// ---- VISUs/SETTING/SettingArm_Page.TcVIS
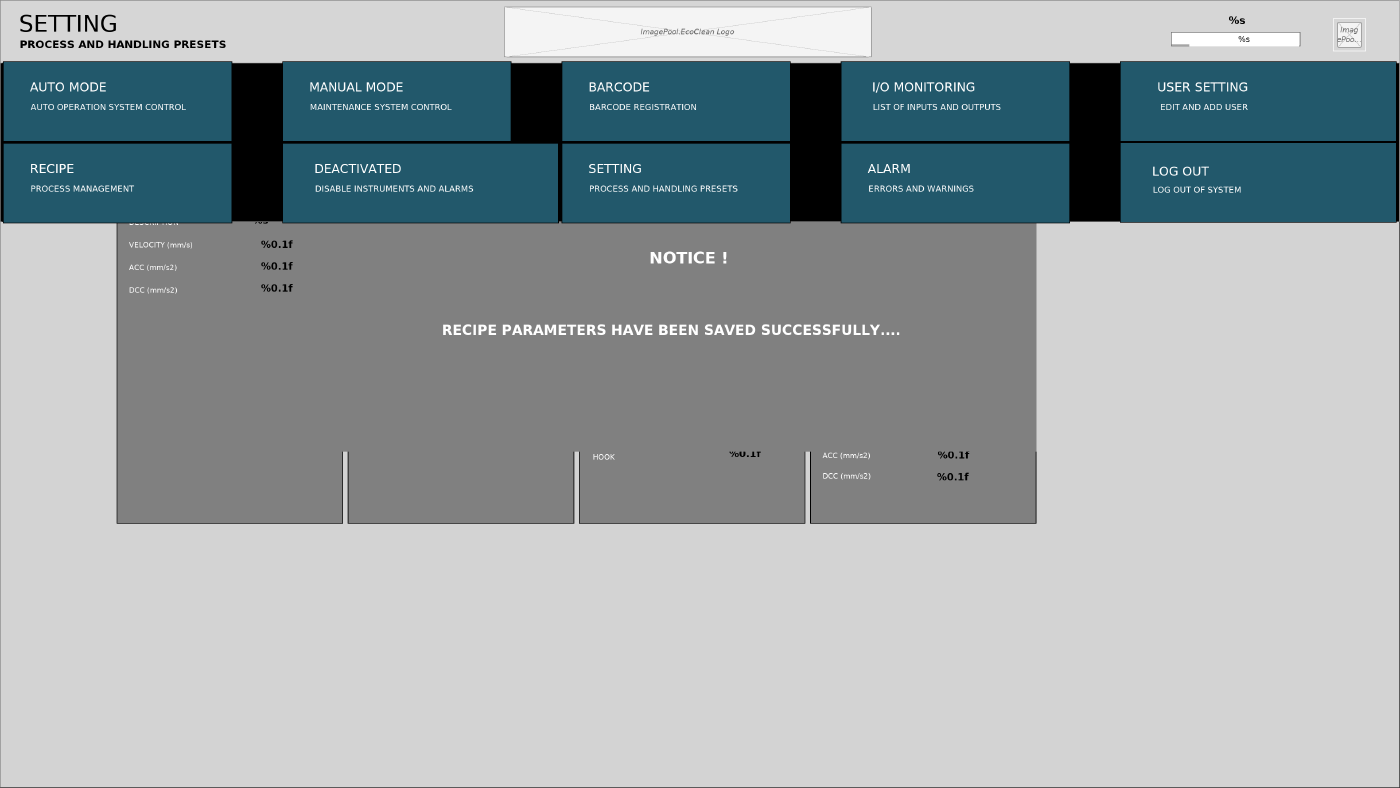
VISUALIZATION SettingArm_Page  // 1920x1081
    Rectangle (0,101 1920x980)
    Rectangle (0,63 1920x26)
        p3528305787: HMI_Ctrl.ANIMATION3
    Rectangle (0,0 1919x85)
    Label (23,6 267x53), "SETTING"
    Label (24,49 320x24), "PROCESS AND HANDLING PRESETS"
    Group (1828,25 45x45)
        OnMouseClick: toggle HMI_Ctrl.MenuButton
        RoundedRectangle (0,0 45x45), colour toggle: HMI_Ctrl.MenuButton
        Image (6,5 33x35), image: ImagePool.Menu Button
    Ellipse (867,123 25x25)
    Ellipse (948,123 25x25)
    Ellipse (904,130 10x10)
    Ellipse (926,130 10x10)
    Ellipse (985,130 10x10)
    Ellipse (1007,130 10x10)
    Ellipse (1029,123 25x25)
    Label (847,153 64x24), "BASIC"
    Label (928,153 64x24), "PROCESS"
    Label (1009,153 64x24), "ARM"
    Image (790,113 45x45), image: ImagePool.Previous Button
        OnMouseClick: change screen: SettingProcess_Page
    RoundedRectangle (1441,125 314x48)
    ComboBoxInteger (1555,132 189x37), variable: iArmSettingStnNoBuffer, text list: 'TextList_Arm_Setting'
    Label (1461,141 79x24), "STATION"
    Rectangle (160,218 310x500)
    Rectangle (160,219 310x27)
    Label (178,222 143x24), "ARM SPEED PROFILE"
    Label (174,262 141x24), "SPEED PROFILE NO."
    Label (174,293 108x24), "DESCRIPTION"
    Label (174,324 116x24), "VELOCITY (mm/s)"
    Label (174,355 118x24), "ACC (mm/s2)"
    Label (174,386 82x24), "DCC (mm/s2)"
    Rectangle (477,218 310x500)
    Rectangle (477,219 310x27)
    Label (495,222 213x24), "ARM UP AND DOWN PATTERN"
    Rectangle (794,218 310x500)
    Rectangle (794,219 310x27)
    Label (812,222 228x24), "ARM VERTICAL POSITION (MM)"
    Rectangle (1111,218 310x500)
    Rectangle (1111,219 310x27)
    Label (1129,222 200x24), "ARM VERTICAL SETTING"
    Label (1125,262 109x24), "1st VELO (mm/s)"
    Label (1125,293 108x24), "ACC (mm/s2)"
    Label (491,262 147x24), "SPEED PATTERN NO"
    Label (491,293 108x24), "DESCRIPTION"
    Label (491,324 196x24), "1ST STAGE SPEED PROFILE"
    Label (491,355 186x24), "2ND STAGE SPEED PROFILE"
    Label (491,391 186x24), "3RD STAGE SPEED PROFILE"
    Label (491,427 186x24), "4TH STAGE SPEED PROFILE"
    Label (808,262 147x24), "TOP POSITION"
    Label (808,293 108x24), "1ST STAGE"
    Label (808,324 196x24), "2ND STAGE"
    Label (808,355 186x24), "3RD STAGE"
    Label (808,386 186x24), "4TH STAGE"
    Label (808,427 186x24), "BOTTOM POSITION"
    Rectangle (1111,539 310x27)
    Label (1129,541 200x24), "ARM HORIZONTAL SETTING"
    Rectangle (310,267 140x17), "%i", text variable: DSA31ArmSpeedProfileStore.iArmSpdProfileNo, input disabled if: bMainOnOff
        OnMouseDown: write the text variable via VisuDialogs.Numpad, min 1, max 20
    Rectangle (263,294 189x17), "%s", text variable: DSA31ArmSpeedProfileStore.DsArmSpeedProfile.sDescription, input disabled if: bMainOnOff
        OnMouseDown: write the text variable via VisuDialogs.Keypad
    Rectangle (310,327 140x17), "%0.1f", text variable: DSA31ArmSpeedProfileStore.DsArmSpeedProfile.lrSpeedVelo, input disabled if: bMainOnOff
        OnMouseDown: write the text variable via VisuDialogs.Numpad, min 2, max 400
    Rectangle (310,357 140x17), "%0.1f", text variable: DSA31ArmSpeedProfileStore.DsArmSpeedProfile.lrAcc, input disabled if: bMainOnOff
        OnMouseDown: write the text variable via VisuDialogs.Numpad, min 100, max 1500
    Rectangle (310,387 140x17), "%0.1f", text variable: DSA31ArmSpeedProfileStore.DsArmSpeedProfile.lrDcc, input disabled if: bMainOnOff
        OnMouseDown: write the text variable via VisuDialogs.Numpad, min 100, max 1500
    Rectangle (653,264 131x17), "%i", text variable: DSA21UpDownPatternStore.iUpDownPatternNo, input disabled if: bMainOnOff
        OnMouseDown: write the text variable via VisuDialogs.Numpad, min 1, max 20
    Rectangle (654,325 129x17), "%i", text variable: DSA21UpDownPatternStore.DsInUpDownPatternMemory.iZone1SpdProfileNo, input disabled if: bMainOnOff
        OnMouseDown: write the text variable via VisuDialogs.Numpad, min 1, max 20
    Rectangle (654,360 129x17), "%i", text variable: DSA21UpDownPatternStore.DsInUpDownPatternMemory.iZone2SpdProfileNo, input disabled if: bMainOnOff
        OnMouseDown: write the text variable via VisuDialogs.Numpad, min 1, max 20
    Rectangle (654,400 129x17), "%i", text variable: DSA21UpDownPatternStore.DsInUpDownPatternMemory.iZone3SpdProfileNo, input disabled if: bMainOnOff
        OnMouseDown: write the text variable via VisuDialogs.Numpad, min 1, max 20
    Rectangle (654,432 129x17), "%i", text variable: DSA21UpDownPatternStore.DsInUpDownPatternMemory.iZone4SpdProfileNo, input disabled if: bMainOnOff
        OnMouseDown: write the text variable via VisuDialogs.Numpad, min 1, max 20
    Rectangle (583,294 189x17), "%s", text variable: DSA21UpDownPatternStore.DsInUpDownPatternMemory.sDescription, input disabled if: bMainOnOff
        OnMouseDown: write the text variable via VisuDialogs.Keypad
    Rectangle (951,264 140x17), "%0.1f", text variable: Arm1TopPos[iArmSettingStnNo], input disabled if: bMainOnOff
        OnMouseDown: write the text variable via VisuDialogs.Numpad
    Rectangle (951,294 140x17), "%0.1f", text variable: Arm1Pos1stStage[iArmSettingStnNo], input disabled if: bMainOnOff
        OnMouseDown: write the text variable via VisuDialogs.Numpad
    Rectangle (951,324 140x17), "%0.1f", text variable: Arm1Pos2ndStage[iArmSettingStnNo], input disabled if: bMainOnOff
        OnMouseDown: write the text variable via VisuDialogs.Numpad
    Rectangle (951,354 140x17), "%0.1f", text variable: Arm1Pos3rdStage[iArmSettingStnNo], input disabled if: bMainOnOff
        OnMouseDown: write the text variable via VisuDialogs.Numpad
    Rectangle (951,389 140x17), "%0.1f", text variable: Arm1Pos4thStage[iArmSettingStnNo], input disabled if: bMainOnOff
        OnMouseDown: write the text variable via VisuDialogs.Numpad
    Rectangle (951,424 140x17), "%0.1f", text variable: Arm1BottomPos[iArmSettingStnNo], input disabled if: bMainOnOff
        OnMouseDown: write the text variable via VisuDialogs.Numpad
    Rectangle (794,539 310x27)
    Label (811,541 228x24), "ARM HORIZONTAL POSITION (MM)"
    Label (810,584 109x24), "UNHOOK"
    Label (810,615 108x24), "HOOK"
    Rectangle (951,584 140x17), "%0.1f", text variable: Arm1UnHookPos[iArmSettingStnNo], input disabled if: bMainOnOff
        OnMouseDown: write the text variable via VisuDialogs.Numpad
    Rectangle (952,614 140x17), "%0.1f", text variable: Arm1HookPos[iArmSettingStnNo], input disabled if: bMainOnOff
        OnMouseDown: write the text variable via VisuDialogs.Numpad
    Label (1125,321 108x24), "DCC (mm/s2)"
    Rectangle (1237,266 140x17), "%0.1f", text variable: ARlrVertPos_In_HighSpeed[1], input disabled if: bMainOnOff
        OnMouseDown: write the text variable via VisuDialogs.Numpad, min 2, max 400
    Rectangle (1238,296 140x17), "%0.1f", text variable: ARlrVertPos_In_Acc[1], input disabled if: bMainOnOff
        OnMouseDown: write the text variable via VisuDialogs.Numpad, min 200, max 1500
    Rectangle (1237,326 140x17), "%0.1f", text variable: ARlrVertPos_In_Dcc[1], input disabled if: bMainOnOff
        OnMouseDown: write the text variable via VisuDialogs.Numpad, min 200, max 1500
    Label (1125,582 109x24), "1st VELO (mm/s)"
    Label (1125,613 108x24), "ACC (mm/s2)"
    Label (1125,641 108x24), "DCC (mm/s2)"
    Rectangle (1237,586 140x17), "%0.1f", text variable: ARlrHorzPos_In_HighSpeed[1], input disabled if: bMainOnOff
        OnMouseDown: write the text variable via VisuDialogs.Numpad, min 50, max 600
    Rectangle (1238,616 140x17), "%0.1f", text variable: ARlrHorzPos_In_Acc[1], input disabled if: bMainOnOff
        OnMouseDown: write the text variable via VisuDialogs.Numpad, min 200, max 1500
    Rectangle (1237,646 140x17), "%0.1f", text variable: ARlrHorzPos_In_Dcc[1], input disabled if: bMainOnOff
        OnMouseDown: write the text variable via VisuDialogs.Numpad, min 200, max 1500
    Image (691,9 504x69), image: ImagePool.EcoClean Logo
    Label (808,465 186x24), "MID POSITION", invisible if: iArmSettingStnNo<>9
    Rectangle (951,469 140x17), "%0.1f", text variable: Arm1MidPos[iArmSettingStnNo], invisible if: iArmSettingStnNo<>9, input disabled if: bMainOnOff
        OnMouseDown: write the text variable via VisuDialogs.Numpad
    Group (1606,17 179x46)
        Button (0,27 177x19), image: VisuSymbols.Symbols.AddUser
        Rectangle (25,28 150x18), "%s", text variable: fbHmiTF1800_UserlevelManagement.dsHmiUserStatus_Active.sLoginName
        Rectangle (2,0 177x22), "%s", text variable: DSLocalSystemTimeML.sCurrentDT24Hr_General
    Group (1439,220 56x80), invisible if: bMainOnOff
        Label (5,52 51x28), "SAVE", invisible if: bMainOnOff
        RoundedRectangle (0,0 55x56), colour toggle: bRecipeSavePb
            tap bRecipeSavePb
        Image (11,5 34x45), image: ImagePool.Save Button
            OnMouseDown: execute { bRecipeSavePb:=1; }
            OnMouseUp: execute { bRecipeSavePb:=0; }
    Frame (457,253 964x366), invisible if: NOT stWritePersistentData.SaveHR
        shows Popup_Parameter_Saved()
    Frame (0,84 1918x221), invisible if: HMI_Ctrl.CloseMenuButton
        shows Popup_MenuPage()
END_VISUALIZATION

// ---- VISUs/SETTING/SettingProcess_Page.TcVIS
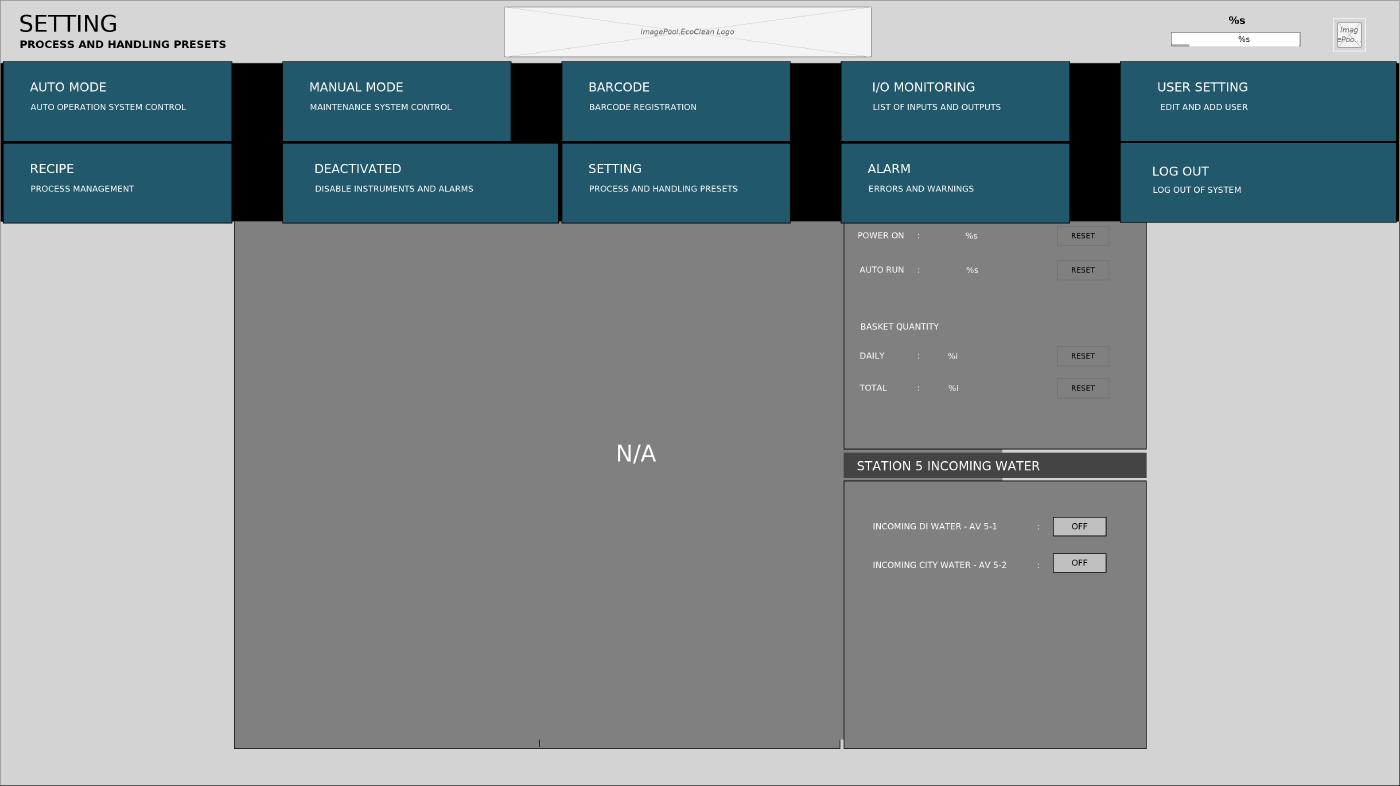
VISUALIZATION SettingProcess_Page  // 1920x1078
    Rectangle (0,101 1920x977)
    Rectangle (321,247 831x780)
    Rectangle (0,63 1920x26)
        p3528305787: HMI_Ctrl.ANIMATION3
    Rectangle (0,0 1919x85)
    Label (23,6 267x53), "SETTING"
    Label (24,49 320x24), "PROCESS AND HANDLING PRESETS"
    Group (1828,25 45x45)
        OnMouseClick: toggle HMI_Ctrl.MenuButton
        RoundedRectangle (0,0 45x45), colour toggle: HMI_Ctrl.MenuButton
        Image (6,5 33x35), image: ImagePool.Menu Button
    Ellipse (867,123 25x25)
    Ellipse (948,123 25x25)
    Ellipse (904,130 10x10)
    Ellipse (926,130 10x10)
    Ellipse (985,130 10x10)
    Ellipse (1007,130 10x10)
    Ellipse (1029,123 25x25)
    Label (847,153 64x24), "BASIC"
    Label (928,153 64x24), "PROCESS"
    Label (1009,153 64x24), "ARM"
    Image (1086,113 45x45), image: ImagePool.Next Button
        OnMouseClick: change screen: SettingArm_Page
    Image (790,113 45x45), image: ImagePool.Previous Button
        OnMouseClick: change screen: Setting_Page
    Rectangle (320,210 833x34)
    Label (582,217 283x24), "TIME OPTIMIZE/TRACKER"
    RoundedRectangle (491,308 30x30), colour toggle: ARbProductRecipeTimeBlockAvailable[1]
    RoundedRectangle (491,378 30x30), colour toggle: ARbProductRecipeTimeBlockAvailable[2]
    RoundedRectangle (491,446 30x30), colour toggle: ARbProductRecipeTimeBlockAvailable[3]
    RoundedRectangle (491,523 30x30), colour toggle: ARbProductRecipeTimeBlockAvailable[4]
    RoundedRectangle (491,598 30x30), colour toggle: ARbProductRecipeTimeBlockAvailable[5]
    RoundedRectangle (491,678 30x30), colour toggle: ARbProductRecipeTimeBlockAvailable[6]
    RoundedRectangle (491,758 30x30), colour toggle: ARbProductRecipeTimeBlockAvailable[7]
    RoundedRectangle (491,829 30x30), colour toggle: ARbProductRecipeTimeBlockAvailable[8]
    RoundedRectangle (491,898 30x30), colour toggle: ARbProductRecipeTimeBlockAvailable[9]
    Label (484,260 103x25), "ENABLE"
    RoundedRectangle (491,968 30x30), colour toggle: ARbProductRecipeTimeBlockAvailable[10]
    Label (385,307 37x24), "1"
    Label (385,377 37x24), "2"
    Label (385,445 37x24), "3"
    Label (385,522 37x24), "4"
    Label (385,597 37x24), "5"
    Label (385,677 37x24), "6"
    Label (385,757 37x24), "7"
    Label (385,828 37x24), "8"
    Label (385,897 37x24), "9"
    Label (380,967 37x24), "10"
    Label (360,248 113x46), "RECIPE NO"
    RoundedRectangle (594,306 90x40), "RESET", input disabled if: bMainOnOff
        tap bTrackerReset[1]
    RoundedRectangle (594,376 90x40), "RESET", input disabled if: bMainOnOff
        tap bTrackerReset[2]
    RoundedRectangle (594,444 90x40), "RESET", input disabled if: bMainOnOff
        tap bTrackerReset[3]
    RoundedRectangle (594,521 90x40), "RESET", input disabled if: bMainOnOff
        tap bTrackerReset[4]
    RoundedRectangle (594,596 90x40), "RESET", input disabled if: bMainOnOff
        tap bTrackerReset[5]
    RoundedRectangle (594,676 90x40), "RESET", input disabled if: bMainOnOff
        tap bTrackerReset[6]
    RoundedRectangle (594,756 90x40), "RESET", input disabled if: bMainOnOff
        tap bTrackerReset[7]
    RoundedRectangle (594,827 90x40), "RESET", input disabled if: bMainOnOff
        tap bTrackerReset[8]
    RoundedRectangle (594,896 90x40), "RESET", input disabled if: bMainOnOff
        tap bTrackerReset[9]
    RoundedRectangle (594,966 90x40), "RESET", input disabled if: bMainOnOff
        tap bTrackerReset[10]
    RoundedRectangle (906,308 30x30), colour toggle: ARbProductRecipeTimeBlockAvailable[11]
    RoundedRectangle (906,378 30x30), colour toggle: ARbProductRecipeTimeBlockAvailable[12]
    RoundedRectangle (906,446 30x30), colour toggle: ARbProductRecipeTimeBlockAvailable[13]
    RoundedRectangle (906,523 30x30), colour toggle: ARbProductRecipeTimeBlockAvailable[14]
    RoundedRectangle (906,598 30x30), colour toggle: ARbProductRecipeTimeBlockAvailable[15]
    RoundedRectangle (906,678 30x30), colour toggle: ARbProductRecipeTimeBlockAvailable[16]
    RoundedRectangle (906,758 30x30), colour toggle: ARbProductRecipeTimeBlockAvailable[17]
    RoundedRectangle (906,829 30x30), colour toggle: ARbProductRecipeTimeBlockAvailable[18]
    RoundedRectangle (906,898 30x30), colour toggle: ARbProductRecipeTimeBlockAvailable[19]
    Label (894,258 103x25), "ENABLE"
    RoundedRectangle (906,968 30x30), colour toggle: ARbProductRecipeTimeBlockAvailable[20]
    Label (803,309 37x24), "11"
    Label (803,379 37x24), "12"
    Label (803,447 37x24), "13"
    Label (803,524 37x24), "14"
    Label (803,599 37x24), "15"
    Label (803,679 37x24), "16"
    Label (803,759 37x24), "17"
    Label (803,830 37x24), "18"
    Label (803,899 37x24), "19"
    Label (802,969 37x24), "20"
    RoundedRectangle (1007,306 90x40), "RESET", input disabled if: bMainOnOff
        tap bTrackerReset[11]
    RoundedRectangle (1007,376 90x40), "RESET", input disabled if: bMainOnOff
        tap bTrackerReset[12]
    RoundedRectangle (1007,444 90x40), "RESET", input disabled if: bMainOnOff
        tap bTrackerReset[13]
    RoundedRectangle (1007,521 90x40), "RESET", input disabled if: bMainOnOff
        tap bTrackerReset[14]
    RoundedRectangle (1007,596 90x40), "RESET", input disabled if: bMainOnOff
        tap bTrackerReset[15]
    RoundedRectangle (1007,676 90x40), "RESET", input disabled if: bMainOnOff
        tap bTrackerReset[16]
    RoundedRectangle (1007,756 90x40), "RESET", input disabled if: bMainOnOff
        tap bTrackerReset[17]
    RoundedRectangle (1007,827 90x40), "RESET", input disabled if: bMainOnOff
        tap bTrackerReset[18]
    RoundedRectangle (1007,896 90x40), "RESET", input disabled if: bMainOnOff
        tap bTrackerReset[19]
    RoundedRectangle (1007,966 90x40), "RESET", input disabled if: bMainOnOff
        tap bTrackerReset[20]
    Label (778,248 113x46), "RECIPE NO"
    Image (691,9 504x69), image: ImagePool.EcoClean Logo
    Rectangle (1050,214 98x26), "ENABLE", colour toggle: bTimeOptimizeDisable, input disabled if: bMainOnOff
        toggle bTimeOptimizeDisable
    Group (1606,17 179x46)
        Button (0,27 177x19), image: VisuSymbols.Symbols.AddUser
        Rectangle (25,28 150x18), "%s", text variable: fbHmiTF1800_UserlevelManagement.dsHmiUserStatus_Active.sLoginName
        Rectangle (2,0 177x22), "%s", text variable: DSLocalSystemTimeML.sCurrentDT24Hr_General
    Line (750,270)
    Line (740,1024) (740,255)
    Group (340,254 783x771), invisible if: bTimeOptimizeDisable
        Rectangle (0,0 1034x760), invisible if: bArmJogEnable
        Label (362,280 341x176), "N/A", invisible if: bArmJogEnable
    Rectangle (1157,248 415x368)
    Rectangle (1157,659 415x368)
    Rectangle (1157,210 415x34)
    Rectangle (1157,621 415x34)
    Label (1242,217 154x24), "MACHINE INFO"
    Label (1174,265 166x24), "MACHINE OPERATION HOUR"
    Label (1173,311 82x24), "POWER ON"
    Label (1176,358 77x24), "AUTO RUN"
    Label (1177,436 134x24), "BASKET QUANTITY"
    Label (1758,515 38x22)
    Rectangle (1248,315 169x17), "%s", text variable: sMachineOnTime_Customer
    Rectangle (1249,362 169x17), "%s", text variable: sMachineRunningTime_Customer
    Label (1176,476 43x24), "DAILY"
    Button (1450,475 71x27), "RESET", colour toggle: bBasketTotalizerResetPB_Daily
        tap bBasketTotalizerResetPB_Daily
    Rectangle (1222,480 169x17), "%i", text variable: diTotalBasketQty_Daily
    Label (1172,627 340x24), "STATION 5 INCOMING WATER"
    Label (1194,710 204x24), "INCOMING DI WATER - AV 5-1"
    Label (1194,763 217x24), "INCOMING CITY WATER - AV 5-2"
    Rectangle (1444,709 73x26), "ON", input disabled if: bMainOnOff
    Rectangle (1444,759 73x26), "ON", input disabled if: bMainOnOff
    Label (1176,520 48x24), "TOTAL"
    Rectangle (1223,524 169x17), "%i", text variable: diTotalBasketQty_Customer
    Button (1450,519 71x27), "RESET", colour toggle: bBasketTotalizerResetPB_Daily
        tap bBasketTotalizerResetPB_User p3779583253=TRUE
    Button (1450,310 71x27), "RESET", colour toggle: bBasketTotalizerResetPB_Daily
        tap bMachineOnTimeRstPB_Customer
    Button (1450,357 71x27), "RESET", colour toggle: bBasketTotalizerResetPB_Daily
        tap bMachineRunningTimeRstPB_Customer
    Rectangle (1444,709 73x26), "OFF", invisible if: ARbOptionSelectedAutoTopupFlag[1], input disabled if: bMainOnOff
        tap ARbOptionSelectedAutoTopupFlag[1]
    Rectangle (1444,759 73x26), "OFF", invisible if: ARbOptionSelectedAutoTopupFlag[2], input disabled if: bMainOnOff
        toggle ARbOptionSelectedAutoTopupFlag[2]
    Label (1255,311 19x24), ":"
    Label (1255,358 19x24), ":"
    Label (1255,476 19x24), ":"
    Label (1255,520 19x24), ":"
    Label (1419,710 19x24), ":"
    Label (1419,763 19x24), ":"
    Frame (0,84 1918x221), invisible if: HMI_Ctrl.CloseMenuButton
        shows Popup_MenuPage()
END_VISUALIZATION

// ---- VISUs/SETTING/Setting_Page.TcVIS
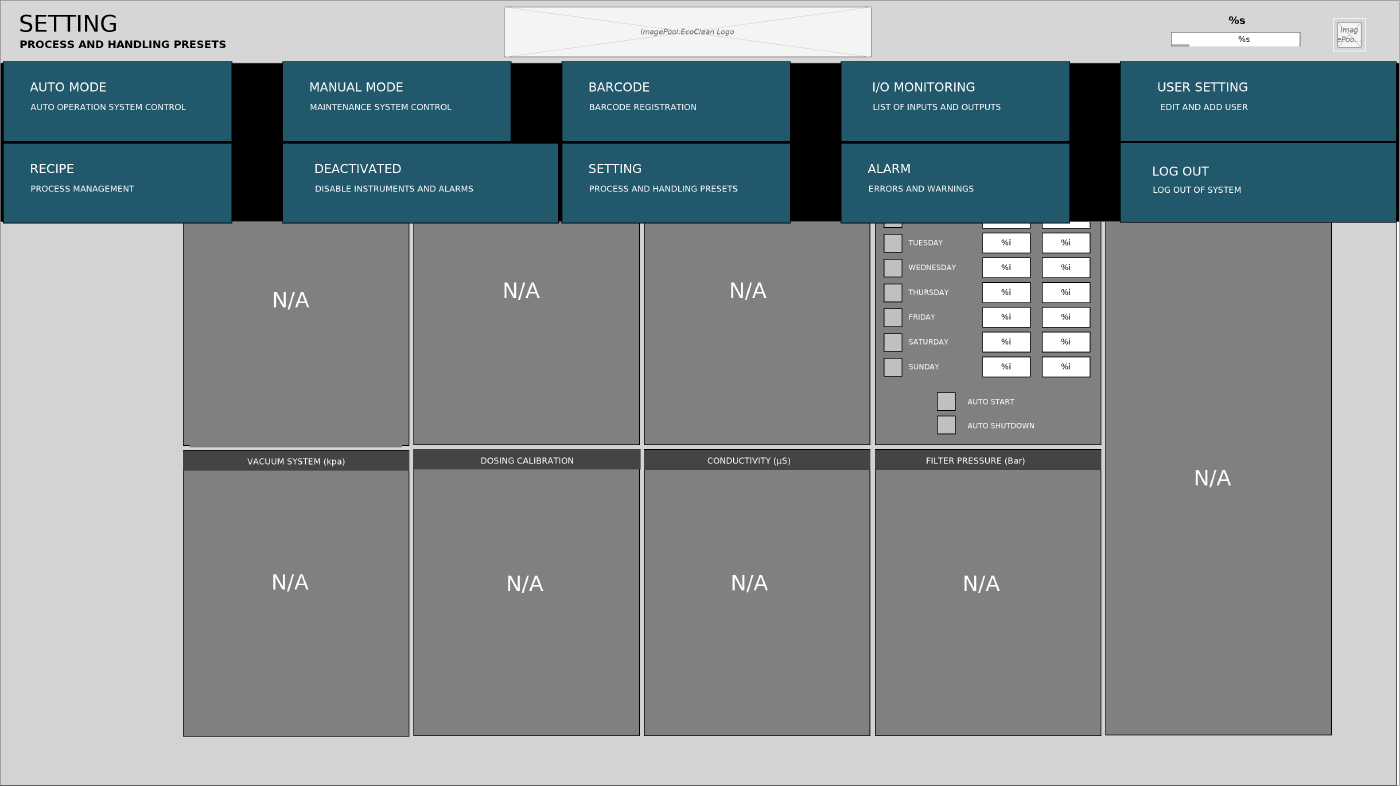
VISUALIZATION Setting_Page  // 1920x1078
    Rectangle (0,98 1915x980)
    Rectangle (0,63 1920x26)
        p3528305787: HMI_Ctrl.ANIMATION3
    Rectangle (0,0 1919x85)
    Label (23,6 267x53), "SETTING"
    Label (24,49 320x24), "PROCESS AND HANDLING PRESETS"
    Group (1828,25 45x45)
        OnMouseClick: toggle HMI_Ctrl.MenuButton
        RoundedRectangle (0,0 45x45), colour toggle: HMI_Ctrl.MenuButton
        Image (6,5 33x35), image: ImagePool.Menu Button
    Ellipse (867,123 25x25)
    Ellipse (948,123 25x25)
    Ellipse (904,130 10x10)
    Ellipse (926,130 10x10)
    Ellipse (985,130 10x10)
    Ellipse (1007,130 10x10)
    Ellipse (1029,123 25x25)
    Label (847,153 64x24), "BASIC"
    Label (928,153 64x24), "PROCESS"
    Label (1009,153 64x24), "ARM"
    Image (1086,113 45x45), image: ImagePool.Next Button
        OnMouseClick: change screen: SettingProcess_Page
    Rectangle (883,218 310x392)
    Rectangle (883,219 310x27)
    Label (967,223 143x24), "TIMER (sec)"
    Label (897,262 153x24), "TEMP NOT READY ALARM", invisible if: iSettingStnNoBuffer=0 OR iSettingStnNoBuffer=8 OR iSettingStnNoBuffer=5 OR iSettingStnNoBuffer=11
    Label (897,293 108x24), "DRIPPING TIME", invisible if: iSettingStnNoBuffer=0 OR iSettingStnNoBuffer=8 OR iSettingStnNoBuffer=11
    Label (897,324 196x24), "BAD BASKET TOLERANCE TIME", invisible if: iSettingStnNoBuffer=0 OR iSettingStnNoBuffer=8 OR iSettingStnNoBuffer=11
    Label (897,355 186x24), "INCOMING VALVE DELAY OFF", invisible if: iSettingStnNoBuffer=0 OR iSettingStnNoBuffer=9 OR iSettingStnNoBuffer=8 OR iSettingStnNoBuffer=6
    Rectangle (1081,265 119x17), "%i", text variable: ARiStnPreparationTempSv[iSettingStnNo], invisible if: iSettingStnNoBuffer=0 OR iSettingStnNoBuffer=8 OR iSettingStnNoBuffer=5 OR iSettingStnNoBuffer=11, input disabled if: bMainOnOff
        OnMouseDown: write the text variable via VisuDialogs.Numpad, min iStnPreparationTempMINsvHMIDisplay, max iStnPreparationTempMAXSVHMIDisplay
    Rectangle (1081,295 119x17), "%i", text variable: ARiStnDippingTimeSV[iSettingStnNo], invisible if: iSettingStnNoBuffer=0 OR iSettingStnNoBuffer=8 OR iSettingStnNoBuffer=11, input disabled if: bMainOnOff
        OnMouseDown: write the text variable via VisuDialogs.Numpad, min 0, max 100
    Rectangle (1081,325 119x17), "%i", text variable: ARiStnToleranceTimeSV[iSettingStnNo], invisible if: iSettingStnNoBuffer=0 OR iSettingStnNoBuffer=8 OR iSettingStnNoBuffer=11, input disabled if: bMainOnOff
        OnMouseDown: write the text variable via VisuDialogs.Numpad, min 0, max 999
    Rectangle (1081,355 119x17), "%i", text variable: ARiStnTopUpDelayOffTimeSV[iSettingStnNo], invisible if: iSettingStnNoBuffer=0 OR iSettingStnNoBuffer=9 OR iSettingStnNoBuffer=8 OR iSettingStnNoBuffer=6, input disabled if: bMainOnOff
        OnMouseDown: write the text variable via VisuDialogs.Numpad, min 0, max 20
    Label (897,385 186x24), "UNLOADING BUZZER", invisible if: iSettingStnNoBuffer<>8
    Rectangle (1081,387 119x17), "%i", text variable: diUnloadingSingleBasketReachedTimer, invisible if: iSettingStnNoBuffer<>8, input disabled if: bMainOnOff
        OnMouseDown: write the text variable via VisuDialogs.Numpad, min 10, max 999
    RoundedRectangle (1278,119 309x48)
    Label (1298,131 79x24), "STATION"
    ComboBoxInteger (1392,125 175x37), variable: iSettingStnNoBuffer, text list: 'TextList_SettingPage'
    Rectangle (1200,218 310x392)
    Rectangle (1200,219 310x27)
    Label (1275,223 161x24), "7 DAYS PREPARATION"
    Label (1243,287 93x24), "MONDAY"
    RoundedRectangle (1347,285 66x28), "%i", text variable: Day1H[OnOffStatus], invisible if: NOT.Day1En[OnOffStatus], input disabled if: bMainOnOff
        OnMouseDown: write the text variable via VisuDialogs.Keypad, min 0, max 23
    Label (1349,261 62x24), "HOUR"
    Label (1429,260 67x24), "MINUTE"
    Label (1243,321 93x24), "TUESDAY"
    Label (1243,355 93x24), "WEDNESDAY"
    Label (1243,389 93x24), "THURSDAY"
    Label (1243,423 93x24), "FRIDAY"
    Label (1243,457 93x24), "SATURDAY"
    Label (1243,491 93x24), "SUNDAY"
    Label (1324,539 93x24), "AUTO START"
    Label (1324,572 120x24), "AUTO SHUTDOWN"
    RoundedRectangle (1347,319 66x28), "%i", text variable: Day2H[OnOffStatus], invisible if: NOT.Day2En[OnOffStatus], input disabled if: bMainOnOff
        OnMouseDown: write the text variable via VisuDialogs.Keypad, min 0, max 23
    RoundedRectangle (1347,353 66x28), "%i", text variable: Day3H[OnOffStatus], invisible if: NOT.Day3En[OnOffStatus], input disabled if: bMainOnOff
        OnMouseDown: write the text variable via VisuDialogs.Keypad, min 0, max 23
    RoundedRectangle (1347,387 66x28), "%i", text variable: Day4H[OnOffStatus], invisible if: NOT.Day4En[OnOffStatus], input disabled if: bMainOnOff
        OnMouseDown: write the text variable via VisuDialogs.Keypad, min 0, max 23
    RoundedRectangle (1347,421 66x28), "%i", text variable: Day5H[OnOffStatus], invisible if: NOT.Day5En[OnOffStatus], input disabled if: bMainOnOff
        OnMouseDown: write the text variable via VisuDialogs.Keypad, min 0, max 23
    RoundedRectangle (1347,455 66x28), "%i", text variable: Day6H[OnOffStatus], invisible if: NOT.Day6En[OnOffStatus], input disabled if: bMainOnOff
        OnMouseDown: write the text variable via VisuDialogs.Keypad, min 0, max 23
    RoundedRectangle (1347,489 66x28), "%i", text variable: Day7H[OnOffStatus], invisible if: NOT.Day7En[OnOffStatus], input disabled if: bMainOnOff
        OnMouseDown: write the text variable via VisuDialogs.Keypad, min 0, max 23
    RoundedRectangle (1429,285 66x28), "%i", text variable: Day1M[OnOffStatus], invisible if: NOT.Day1En[OnOffStatus], input disabled if: bMainOnOff
        OnMouseDown: write the text variable via VisuDialogs.Keypad, min 0, max 59
    RoundedRectangle (1429,319 66x28), "%i", text variable: Day2M[OnOffStatus], invisible if: NOT.Day2En[OnOffStatus], input disabled if: bMainOnOff
        OnMouseDown: write the text variable via VisuDialogs.Keypad, min 0, max 59
    RoundedRectangle (1429,353 66x28), "%i", text variable: Day3M[OnOffStatus], invisible if: NOT.Day3En[OnOffStatus], input disabled if: bMainOnOff
        OnMouseDown: write the text variable via VisuDialogs.Keypad, min 0, max 59
    RoundedRectangle (1429,387 66x28), "%i", text variable: Day4M[OnOffStatus], invisible if: NOT.Day4En[OnOffStatus], input disabled if: bMainOnOff
        OnMouseDown: write the text variable via VisuDialogs.Keypad, min 0, max 59
    RoundedRectangle (1429,421 66x28), "%i", text variable: Day5M[OnOffStatus], invisible if: NOT.Day5En[OnOffStatus], input disabled if: bMainOnOff
        OnMouseDown: write the text variable via VisuDialogs.Keypad, min 0, max 59
    RoundedRectangle (1429,455 66x28), "%i", text variable: Day6M[OnOffStatus], invisible if: NOT.Day6En[OnOffStatus], input disabled if: bMainOnOff
        OnMouseDown: write the text variable via VisuDialogs.Keypad, min 0, max 59
    RoundedRectangle (1429,489 66x28), "%i", text variable: Day7M[OnOffStatus], invisible if: NOT.Day7En[OnOffStatus], input disabled if: bMainOnOff
        OnMouseDown: write the text variable via VisuDialogs.Keypad, min 0, max 59
    Rectangle (1212,287 25x25), colour toggle: Day1En[OnOffStatus], input disabled if: bMainOnOff
        toggle Day1En[OnOffStatus]
    Rectangle (1212,321 25x25), colour toggle: Day2En[OnOffStatus], input disabled if: bMainOnOff
        toggle Day2En[OnOffStatus]
    Rectangle (1212,355 25x25), colour toggle: Day3En[OnOffStatus], input disabled if: bMainOnOff
        toggle Day3En[OnOffStatus]
    Rectangle (1212,389 25x25), colour toggle: Day4En[OnOffStatus], input disabled if: bMainOnOff
        toggle Day4En[OnOffStatus]
    Rectangle (1212,423 25x25), colour toggle: Day5En[OnOffStatus], input disabled if: bMainOnOff
        toggle Day5En[OnOffStatus]
    Rectangle (1212,457 25x25), colour toggle: Day6En[OnOffStatus], input disabled if: bMainOnOff
        toggle Day6En[OnOffStatus]
    Rectangle (1212,491 25x25), colour toggle: Day7En[OnOffStatus], input disabled if: bMainOnOff
        toggle Day7En[OnOffStatus]
    Rectangle (1285,538 25x25), colour toggle: OnOffStatus=1
        OnMouseDown: execute { OnOffStatus:=1; }
    Rectangle (1285,570 25x25), colour toggle: OnOffStatus=2
        OnMouseDown: execute { OnOffStatus:=2; }
    Rectangle (567,616 310x393)
    Label (582,667 167x28), "CALIBRATE FEED (pulse)"
    Rectangle (779,665 82x28), "%i", text variable: ARDSProminentDosingHMI[iSettingStnNo].In_iCalibrateFeed_Pulse, input disabled if: bMainOnOff
        OnMouseDown: write the text variable via VisuDialogs.Numpad, min 10, max 999
    Label (586,707 159x28), "CALIBRATE RESULT (ml)"
    Rectangle (779,705 82x28), "%i", text variable: ARDSProminentDosingHMI[iSettingStnNo].In_iCalibrateTotalVolumeResult_ml, input disabled if: bMainOnOff
        OnMouseDown: write the text variable via VisuDialogs.Numpad, min 1, max 9999
    Label (586,747 159x28), "CALIBRATE START"
    Rectangle (757,748 110x30), "START", colour toggle: ARDSProminentDosingHMI[iSettingStnNo].In_bCalibratePB, input disabled if: bMainOnOff
        toggle ARDSProminentDosingHMI[iSettingStnNo].In_bCalibratePB
    Rectangle (773,886 74x30), "RESET", colour toggle: ARDSProminentDosingHMI[iSettingStnNo].In_bResetRemainedDosingVolumePB, input disabled if: bMainOnOff
        tap ARDSProminentDosingHMI[HMI_Ctrl.StationInfoPageNo].In_bResetRemainedDosingVolumePB
    Label (588,888 129x28), "RESET REMAINING DOSING VOLUME (ml)"
    Label (586,797 159x28), "CALIBRATE IN PROGRESS"
    Label (586,837 159x28), "CALIBRATE DONE"
    Ellipse (807,795 25x25), colour toggle: ARDSProminentDosingHMI[iSettingStnNo].Out_bCalibrateInProgress
    Ellipse (807,835 25x25), colour toggle: ARDSProminentDosingHMI[iSettingStnNo].Out_bCalibrateDone
    Group (581,653 291x349), invisible if: iSettingStnNoBuffer<>0 AND iSettingStnNoBuffer<>5 AND iSettingStnNoBuffer<>6 AND iSettingStnNoBuffer<>7 AND iSettingStnNoBuffer<>8 AND iSettingStnNoBuffer<>9
        Rectangle (0,0 291x349)
        Label (110,122 81x51), "N/A"
    Rectangle (568,616 310x27)
    Label (635,618 176x28), "DOSING CALIBRATION"
    Rectangle (567,218 310x392)
    Rectangle (567,219 310x27)
    Label (651,221 143x28), "DOSING"
    Label (581,262 129x28), "DOSE PER PULSE (ml)"
    Label (581,299 159x28), "VOLUME PER BASKET (ml)"
    Label (581,336 224x28), "NUMBER OF BASKET BETWEEN DOSING"
    Label (584,373 118x28), "REMAINING DOSING VOLUME (ml)"
    Label (581,460 91x28), "FIRST FILL (ml)"
    Rectangle (768,261 82x28), "%0.02f", text variable: ARDSProminentDosingHMI[iSettingStnNo].In_rVolumePerPulse_ml, input disabled if: bMainOnOff
    Rectangle (768,301 82x28), "%i", text variable: ARDSProminentDosingHMI[iSettingStnNo].In_iVolumePerBasket_ml, input disabled if: bMainOnOff
        OnMouseDown: write the text variable via VisuDialogs.Numpad, min 1, max 9999
    Rectangle (768,331 82x28), "%i", text variable: ARDSProminentDosingHMI[iSettingStnNo].In_iNoOfBasketBetweenAutoDosing, input disabled if: bMainOnOff
        OnMouseDown: write the text variable via VisuDialogs.Numpad, min 1, max 999
    Rectangle (770,369 82x28), "%0.01f", text variable: ARDSProminentDosingHMI[iSettingStnNo].Out_rRemainedDosingVolume_ml
    Rectangle (768,458 82x28), "%i", text variable: ARDSProminentDosingHMI[iSettingStnNo].in_iFirstFillDosing_ml, input disabled if: bMainOnOff
        OnMouseDown: write the text variable via VisuDialogs.Numpad, min 1, max 32767
    Label (584,424 118x28), "TOTALIZER DOSING VOLUME"
    Rectangle (803,420 70x28), "%i", text variable: ARDSProminentDosingHMI[iSettingStnNo].Out_iDosingTotalizer_ml
    Label (581,501 129x28), "RESET REMAINING DOSING VOLUME (ml)"
    Rectangle (768,499 74x30), "RESET", colour toggle: ARDSProminentDosingHMI[iSettingStnNo].In_bResetRemainedDosingVolumePB, input disabled if: bMainOnOff
        tap ARDSProminentDosingHMI[iSettingStnNo].In_bResetRemainedDosingVolumePB
    Label (580,551 152x28), "RESET REMAINING DOSING TOTALIZER (ml)"
    Rectangle (767,549 74x30), "RESET", colour toggle: ARDSProminentDosingHMI[iSettingStnNo].In_bResetDosingTotalizerPB, input disabled if: bMainOnOff
        tap ARDSProminentDosingHMI[iSettingStnNo].In_bResetDosingTotalizerPB
    Rectangle (883,616 310x393)
    Rectangle (883,617 310x27)
    Label (967,620 143x24), "CONDUCTIVITY (μS)"
    Label (896,661 108x24), "ACTUAL VALUE"
    Rectangle (1018,662 169x17), "%0.01f", text variable: ARrStnConductivityPV[iSettingStnNo]
    Rectangle (1018,693 169x17), "%0.01f", text variable: ARrStnLowConductivitySv[iSettingStnNo], input disabled if: bMainOnOff
        OnMouseDown: write the text variable via VisuDialogs.Numpad, min 0, max 999
    Rectangle (1018,723 169x17), "%0.01f", text variable: ARrStnHighConductivitySv[iSettingStnNo], input disabled if: bMainOnOff
        OnMouseDown: write the text variable via VisuDialogs.Numpad, min 0, max 99999
    Rectangle (895,692 119x17), "LOW ALARM", text variable: sDisplayConductivity[1]
    Rectangle (895,722 119x17), "HIGH ALARM", text variable: sDisplayConductivity[2]
    Group (889,652 291x349), invisible if: iSettingStnNoBuffer=5
        Rectangle (0,0 291x349)
        Label (110,122 81x51), "N/A"
    Rectangle (1200,616 310x393)
    Rectangle (1200,617 310x27)
    Label (1267,620 177x24), "FILTER PRESSURE (Bar)"
    Label (1212,661 108x24), "ACTUAL VALUE"
    Rectangle (1334,662 169x17), "%0.01f", text variable: ARrStnFilterPressurePV[iSettingStnNo]
    Rectangle (1334,693 169x17), "%0.01f", text variable: ARrStnLowFilterPressureSv[iSettingStnNo], input disabled if: bMainOnOff
        OnMouseDown: write the text variable via VisuDialogs.Numpad, min 0, max 999
    Rectangle (1334,723 169x17), "%0.01f", text variable: ARrStnHighFilterPressureSv[iSettingStnNo], input disabled if: bMainOnOff
        OnMouseDown: write the text variable via VisuDialogs.Numpad, min 0, max 999
    Label (1212,691 108x24), "LOW ALARM"
    Label (1212,720 108x24), "HIGH ALARM"
    Group (1207,653 291x349), invisible if: iSettingStnNoBuffer<> 6 AND iSettingStnNoBuffer<> 7 AND iSettingStnNoBuffer<> 8 AND iSettingStnNoBuffer<> 9
        Rectangle (0,0 291x349)
        Label (110,122 81x51), "N/A"
    Rectangle (251,218 310x393)
    Rectangle (251,219 310x27)
    Label (315,223 183x24), "TANK TEMPERATURE (°C)"
    Label (265,262 109x24), "SET VALUE", invisible if: iSettingStnNoBuffer=5
    Label (265,293 108x24), "ACTUAL VALUE"
    Label (265,324 116x24), "HIGH TEMP ALARM", invisible if: iSettingStnNoBuffer=5
    Label (265,355 133x24), "1ST LIMIT ALARM (+/-)", invisible if: iSettingStnNoBuffer=5
    Label (265,385 82x24), "HYSTERESIS", invisible if: iSettingStnNoBuffer=5
    Label (265,416 82x24), "READY (+/-)", invisible if: iSettingStnNoBuffer=5
    Rectangle (387,266 169x17), "%0.01f", text variable: ARrStnTempSV[iSettingStnNo], invisible if: iSettingStnNoBuffer=5, input disabled if: bMainOnOff
        OnMouseDown: write the text variable via VisuDialogs.Numpad, min rStnTempMINsvHMIDisplay, max rStnTempMAXsvHMIDisplay
    Rectangle (387,297 169x17), "%0.01f", text variable: ARrStnTempPV[iSettingStnNo]
    Rectangle (387,328 169x17), "%0.01f", text variable: ARrStnTempHALsv[iSettingStnNo], invisible if: iSettingStnNoBuffer=5, input disabled if: bMainOnOff
        OnMouseDown: write the text variable via VisuDialogs.Numpad, min rStnTempHALMINsvHMIDisplay, max rStnTempHALMAXsvHMIDisplay
    Rectangle (387,359 169x17), "%0.01f", text variable: ARrStnTemp1stLimitSv[iSettingStnNo], invisible if: iSettingStnNoBuffer=5, input disabled if: bMainOnOff
        OnMouseDown: write the text variable via VisuDialogs.Numpad, min rStnTemp1stLimitMINsvHMIDisplay, max rStnTemp1stLimitMAXsvHMIDisplay
    Rectangle (387,389 169x17), "%0.01f", text variable: ARrStnTempHYSsv[iSettingStnNo], invisible if: iSettingStnNoBuffer=5, input disabled if: bMainOnOff
        OnMouseDown: write the text variable via VisuDialogs.Numpad, min rStnTempHYSMINsvHMIDisplay, max rStnTempHYSMAXsvHMIDisplay
    Rectangle (387,420 169x17), "%0.01f", text variable: ARrStnTempRDYsv[iSettingStnNo], invisible if: iSettingStnNoBuffer=5, input disabled if: bMainOnOff
        OnMouseDown: write the text variable via VisuDialogs.Numpad, min rStnTempRDYMINsvHMIDisplay, max rStnTempRDYMAXsvHMIDisplay
    Group (260,264 291x332), invisible if: iSettingStnNoBuffer<>7 AND iSettingStnNoBuffer<>8 AND iSettingStnNoBuffer<>9
        Rectangle (0,0 291x349)
        Label (110,122 81x51), "N/A"
    Rectangle (251,617 310x393)
    Rectangle (251,618 310x27)
    Label (298,621 217x24), "VACUUM SYSTEM (kpa)"
    Image (691,9 504x69), image: ImagePool.EcoClean Logo
    Group (1606,17 179x46)
        Button (0,27 177x19), image: VisuSymbols.Symbols.AddUser
        Rectangle (25,28 150x18), "%s", text variable: fbHmiTF1800_UserlevelManagement.dsHmiUserStatus_Active.sLoginName
        Rectangle (2,0 177x22), "%s", text variable: DSLocalSystemTimeML.sCurrentDT24Hr_General
    Rectangle (720,420 82x28), "%i", text variable: ARDSProminentDosingHMI[iSettingStnNo].Out_iDosingTotalizer_Litre
    Label (756,398 24x28), "L"
    Label (821,398 24x28), "ml"
    Group (576,251 291x346), invisible if: iSettingStnNoBuffer<>0 AND iSettingStnNoBuffer<>5 AND iSettingStnNoBuffer<>6 AND iSettingStnNoBuffer<>7 AND iSettingStnNoBuffer<>8 AND iSettingStnNoBuffer<>9
        Rectangle (0,0 291x349)
        Label (110,122 81x51), "N/A"
    Group (887,251 291x346), invisible if: iSettingStnNoBuffer<>0 AND iSettingStnNoBuffer<>7 AND iSettingStnNoBuffer<>9
        Rectangle (0,0 291x349)
        Label (110,122 81x51), "N/A"
    Label (267,661 108x24), "VACUUM LEVEL"
    Rectangle (389,662 169x17), "%0.01f", text variable: ARrStnVacuumPV[iSettingStnNo]
    Rectangle (389,693 169x17), "%0.01f", text variable: ARrStnHighVacuumLevelSV[iSettingStnNo], input disabled if: bMainOnOff
        OnMouseDown: write the text variable via VisuDialogs.Numpad, min -120, max 10
    Rectangle (389,723 169x17), "%0.01f", text variable: ARrStnLowVacuumLevelSV[iSettingStnNo], input disabled if: bMainOnOff
        OnMouseDown: write the text variable via VisuDialogs.Numpad, min -120, max 10
    Rectangle (266,692 119x17), "HIGH VACUUM LEVEL", text variable: sDisplayConductivity[1]
    Rectangle (266,722 119x17), "LOW VACUUM LEVEL", text variable: sDisplayConductivity[2]
    Group (259,651 291x349), invisible if: iSettingStnNoBuffer= 6
        Rectangle (0,0 291x349)
        Label (110,122 81x51), "N/A"
    Rectangle (1516,218 310x790)
    Rectangle (1516,219 310x27)
    Label (1558,223 233x24), "VACUUM PUMP SERVICE ROUTINE"
    Label (1530,263 177x24), "VACUUM PUMP SERVICE HOUR"
    Rectangle (1741,327 58x17), "%i", text variable: ARdiVacPump2ndLimitTimerSV[iSettingStnNo], input disabled if: iCurrentUserGroupID<6 OR bMainOnOff
        OnMouseDown: write the text variable via VisuDialogs.Numpad, min 0, max 999
    Label (1530,321 92x24), "2nd LIMIT TIMER"
    Label (1530,383 159x24), "VACUUM PUMP TIMER"
    Rectangle (1745,379 57x24), "RESET", colour toggle: ARDSProminentDosingHMI[iSettingStnNo].In_bResetRemainedDosingVolumePB, input disabled if: iCurrentUserGroupID<6 OR bMainOnOff
        tap ARbVacuumPumpTimerReset[iSettingStnNo]
    Label (1530,349 159x24), "VACUUM PUMP RUN TIMER"
    Rectangle (1731,353 78x17), "%s", text variable: ARsVacuumPumpRunningTime[iSettingStnNo]
    Label (1530,293 92x24), "1st LIMIT TIMER"
    Rectangle (1741,299 58x17), "%i", text variable: ARdiVacPump1stLimitTimerSV[iSettingStnNo], input disabled if: iCurrentUserGroupID<6 OR bMainOnOff
        OnMouseDown: write the text variable via VisuDialogs.Numpad, min 0, max 999
    Label (1530,433 248x24), "VACUUM PUMP ROUTINE SERVICE DAYS"
    Rectangle (1741,497 58x17), "%i", text variable: ARiAlarmDaysSV_Routine[iSettingStnNo], input disabled if: iCurrentUserGroupID<6 OR bMainOnOff
        OnMouseDown: write the text variable via VisuDialogs.Numpad, min 0, max 999
    Label (1530,491 92x24), "2nd LIMIT TIMER"
    Label (1530,553 159x24), "VACUUM PUMP TIMER"
    Rectangle (1745,549 57x24), "RESET", colour toggle: ARDSProminentDosingHMI[iSettingStnNo].In_bResetRemainedDosingVolumePB, input disabled if: iCurrentUserGroupID<6 OR bMainOnOff
        tap ARbDaysPvReset_Routine[6]
    Label (1530,519 159x24), "VACUUM PUMP RUN TIMER"
    Rectangle (1731,523 78x17), "%i", text variable: ARiRunDaysPV_Routine[iSettingStnNo]
    Label (1530,463 92x24), "1st LIMIT TIMER"
    Rectangle (1741,469 58x17), "%i", text variable: ARiWarningDaysSV_Routine[iSettingStnNo], input disabled if: iCurrentUserGroupID<6 OR bMainOnOff
        OnMouseDown: write the text variable via VisuDialogs.Numpad, min 0, max 999
    Label (1530,613 227x24), "VACUUM PUMP MAJOR SERVICE DAYS"
    Rectangle (1741,677 58x17), "%i", text variable: ARiAlarmDaysSV_Major[iSettingStnNo], input disabled if: iCurrentUserGroupID<6 OR bMainOnOff
        OnMouseDown: write the text variable via VisuDialogs.Numpad, min 0, max 999
    Label (1530,671 92x24), "2nd LIMIT TIMER"
    Label (1530,733 159x24), "VACUUM PUMP TIMER"
    Rectangle (1745,729 57x24), "RESET", colour toggle: ARDSProminentDosingHMI[iSettingStnNo].In_bResetRemainedDosingVolumePB, input disabled if: iCurrentUserGroupID<6 OR bMainOnOff
        tap ARbDaysPvReset_Major[6]
    Label (1530,699 159x24), "VACUUM PUMP RUN TIMER"
    Rectangle (1731,703 78x17), "%i", text variable: ARiRunDaysPV_Major[iSettingStnNo]
    Label (1530,643 92x24), "1st LIMIT TIMER"
    Rectangle (1741,649 58x17), "%i", text variable: ARiWarningDaysSV_Major[iSettingStnNo], input disabled if: iCurrentUserGroupID<6 OR bMainOnOff
        OnMouseDown: write the text variable via VisuDialogs.Numpad, min 0, max 999
    Group (1526,259 283x735), invisible if: iSettingStnNoBuffer=6
        Rectangle (0,0 283x735)
        Label (108,372 74x49), "N/A"
    Frame (0,84 1918x221), invisible if: HMI_Ctrl.CloseMenuButton
        shows Popup_MenuPage()
END_VISUALIZATION

// ---- VISUs/TextList_1_20.TcTLO
TEXTLIST TextList_1_20
  1 = '1'
  2 = '2'
  3 = '3'
  4 = '4'
  5 = '5'
  6 = '6'
  7 = '7'
  8 = '8'
  9 = '9'
  10 = '10'
  11 = '11'
  12 = '12'
  13 = '13'
  14 = '14'
  15 = '15'
  16 = '16'
  17 = '17'
  18 = '18'
  19 = '19'
  20 = '20'
  0 = '0'
   = ''
END_TEXTLIST

// ---- VISUs/TextList_1_20_Speed.TcTLO
TEXTLIST TextList_1_20_Speed
  1 = '1'
  2 = '2'
  3 = '3'
  4 = '4'
  5 = '5'
  6 = '6'
  7 = '7'
  8 = '8'
  9 = '9'
  10 = '10'
  11 = '11'
  12 = '12'
  13 = '13'
  14 = '14'
  15 = '15'
  16 = '16'
  17 = '17'
  18 = '18'
  19 = '19'
  20 = '20'
   = ''
END_TEXTLIST

// ---- VISUs/TextList_AccessLevel.TcTLO
TEXTLIST TextList_AccessLevel
  0 = 'GUEST'
  1 = 'OPERATOR'
  2 = 'TECHNICIAN'
  3 = 'ENGINEER'
  4 = 'MANAGER'
  5 = 'JKS'
   = ''
END_TEXTLIST

// ---- VISUs/TextList_Arm_Setting.TcTLO
TEXTLIST TextList_Arm_Setting
  1 = '1'
  2 = '2'
  3 = '3'
  4 = '4'
  5 = '5'
  6 = '6'
  7 = 'LOADING'
  8 = 'UNLOADING'
   = ''
END_TEXTLIST

// ---- VISUs/TextList_ManualPage.TcTLO
TEXTLIST TextList_ManualPage
  0 = 'GENERAL'
  1 = '1'
  2 = '2'
  3 = '3'
  4 = '4'
  5 = '5'
  6 = '6'
  7 = 'LOADING'
   = ''
END_TEXTLIST

// ---- VISUs/TextList_Recipe.TcTLO
TEXTLIST TextList_Recipe
  1 = '1'
  2 = '2'
  3 = '3'
  4 = '4'
  5 = '5'
  6 = '6'
   = ''
END_TEXTLIST

// ---- VISUs/TextList_SettingPage.TcTLO
TEXTLIST TextList_SettingPage
  1 = '1'
  2 = '2'
  3 = '3'
  4 = '4'
  5 = '5'
  6 = '6'
  7 = 'LOADING'
  8 = 'UNLOADING'
  9 = 'GENERAL'
   = ''
END_TEXTLIST

// ---- VISUs/TextList_SettingPage_2.TcTLO
TEXTLIST TextList_SettingPage_2
  1 = 'STATION 01'
  2 = 'STATION 02'
  3 = 'STATION 03'
  4 = 'STATION 04'
  5 = 'STATION 05'
  6 = 'STATION 06'
  7 = 'LOADING'
  8 = 'UNLOADING'
  9 = 'GENERAL'
   = ''
END_TEXTLIST

// ---- VISUs/TextList_StationInfoPage.TcTLO
TEXTLIST TextList_StationInfoPage
  1 = '1'
  2 = '2'
  3 = '3'
  4 = '4'
  5 = '5'
  6 = '6'
  10 = 'LOADING'
  11 = 'UNLOADING'
  13 = 'GENERAL'
   = ''
END_TEXTLIST

// ---- VISUs/USER_LOGIN/Login_Page.TcVIS
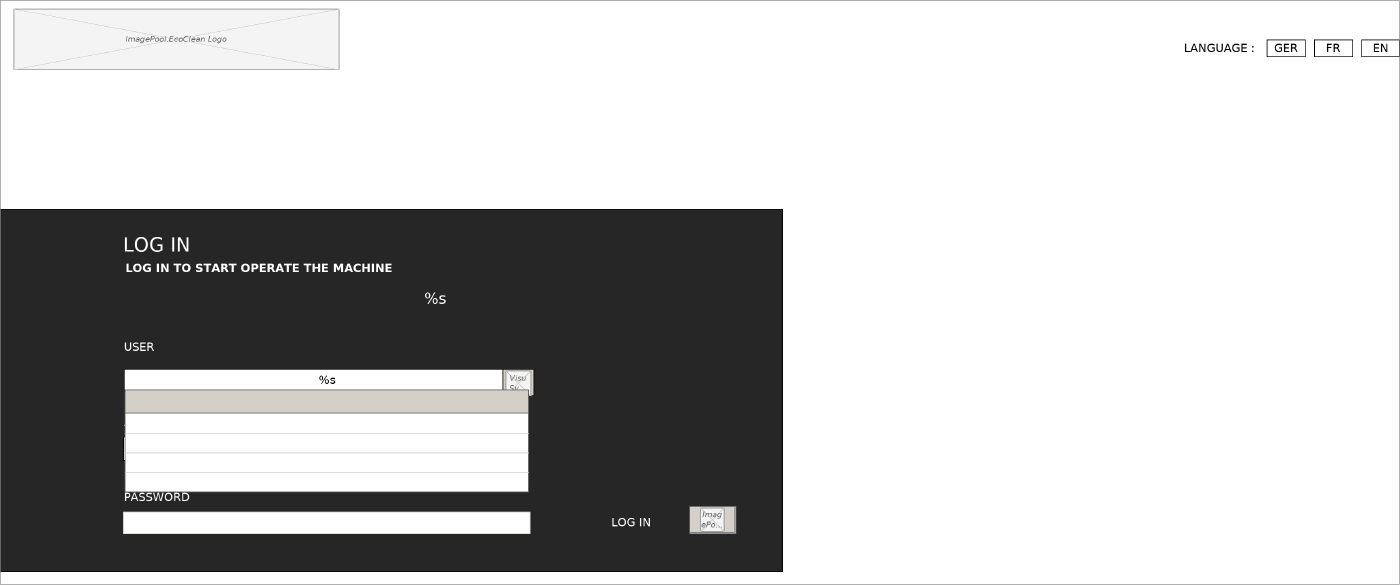
VISUALIZATION Login_Page  // 1775x742
    Label (1498,52 112x18), "LANGUAGE :"
    Rectangle (1606,50 49x22), "GER"
        OnMouseDown: ChangeLanguage ChangeLanguage=German
    Rectangle (0,252 1x490)
        p3528305787: HMI_Ctrl.ANIMATION2
    Rectangle (0,265 992x460)
    Label (153,284 221x53), "LOG IN"
    Label (156,321 609x38), "LOG IN TO START OPERATE THE MACHINE"
    Label (154,604 216x53), "PASSWORD"
    Textfield (156,649 516x28), text variable: sPasswordField
        OnMouseDown: write the text variable via Default, password
    Label (154,409 123x62), "USER"
    Label (154,509 216x53), "ACCESS LEVEL"
    Group (874,642 59x35)
        toggle bLoginPB
        Button (0,0 59x35)
        Image (14,2 30x30), image: ImagePool.Log In
    Label (733,639 135x47), "LOG IN"
    Group (157,468 516x28)
        toggle bUserNameLoginPageOn
        Rectangle (0,0 516x28), "%s", text variable: fbHmiTF1800_UserlevelManagement.dsHmiUserReg.ARsLoginName[iLoginNameId]
        Group (480,0 35x28)
            Rectangle (0,0 40x34)
            Image (4,2 32x32), image: VisuSymbols.Symbols.TriangleDown
    Textfield (168,364 768x30), "%s", text variable: sMessage
    Rectangle (156,554 513x30), "%s", text variable: fbHmiTF1800_UserlevelManagement.dsHmiUserReg.ARwsUserGroupName[iLoginNameId]
    Table (158,494 512x130), invisible if: NOT bUserNameLoginPageOn, data array: fbHmiTF1800_UserlevelManagement.dsHmiUserReg.ARsLoginName
        p3854506369: fbHmiTF1800_UserlevelManagement.dsHmiUserReg.ARsLoginName[INDEX]
        p2232123230: Login Name
        p1137915858: iLoginNameId
        Columns.Column.[0].Template: toggle bUserNameLoginPageOn
    Image (17,11 413x77), image: ImagePool.EcoClean Logo
    Rectangle (1666,50 49x22), "FR"
        OnMouseDown: ChangeLanguage ChangeLanguage=France
    Rectangle (1726,50 49x22), "EN"
        OnMouseDown: ChangeLanguage ChangeLanguage=English
END_VISUALIZATION

// ---- VISUs/USER_SETTING/AddNewUser_Page.TcVIS
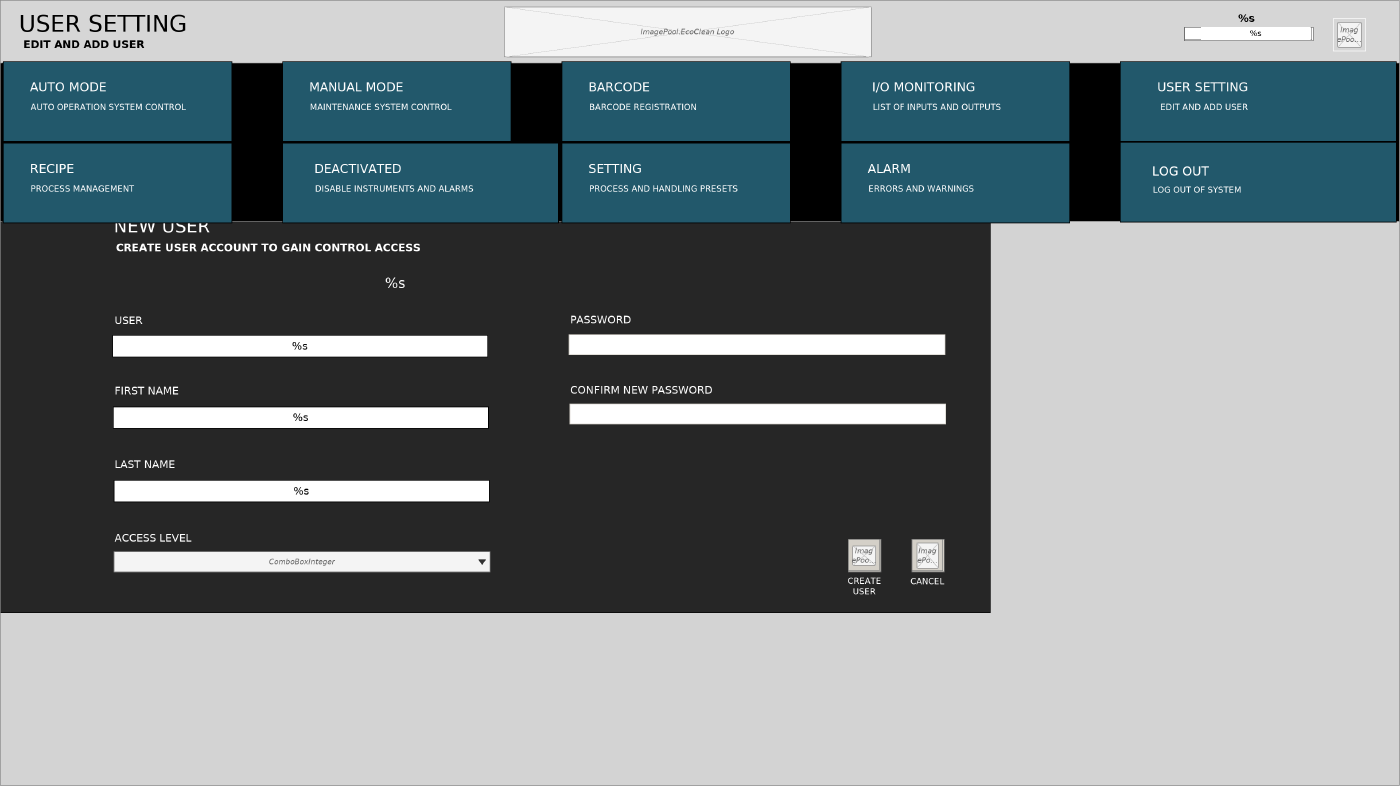
VISUALIZATION AddNewUser_Page  // 1920x1079
    Rectangle (0,98 1920x981)
    Rectangle (0,63 1920x26)
        p3528305787: HMI_Ctrl.ANIMATION3
    Rectangle (0,0 1919x85)
    Label (23,6 310x53), "USER SETTING"
    Label (29,49 320x24), "EDIT AND ADD USER"
    Group (1828,25 45x45)
        OnMouseClick: toggle HMI_Ctrl.MenuButton
        RoundedRectangle (0,0 45x45), colour toggle: HMI_Ctrl.MenuButton
        Image (6,5 33x35), image: ImagePool.Menu Button
    Image (691,9 504x69), image: ImagePool.EcoClean Logo
    Group (1621,14 180x42)
        Rectangle (0,0 177x22), "%s", text variable: DSLocalSystemTimeML.sCurrentDT24Hr_General
        Button (3,23 177x19), image: VisuSymbols.Symbols.AddUser
        Rectangle (26,23 150x18), "%s", text variable: fbHmiTF1800_UserlevelManagement.dsHmiUserStatus_Active.sLoginName
    Rectangle (0,264 1358x577)
    Label (153,284 221x53), "NEW USER"
    Label (156,321 609x38), "CREATE USER ACCOUNT TO GAIN CONTROL ACCESS"
    Label (154,712 216x53), "ACCESS LEVEL"
    ComboBoxInteger (156,757 516x28), variable: sUM_NewUserGroupId, text list: 'TextList_AccessLevel'
    Label (154,611 216x53), "LAST NAME"
    Label (154,409 123x62), "USER"
    Label (154,510 216x53), "FIRST NAME"
    Label (779,408 195x62), "PASSWORD"
    Label (779,509 229x53), "CONFIRM NEW PASSWORD"
    Textfield (781,554 516x28), text variable: sUM_ConfirmPassword
        OnMouseDown: write the text variable via Default, password
    Textfield (780,459 516x28), text variable: sUM_NewPassword
        OnMouseDown: write the text variable via Default, password
    RoundedRectangle (601,151 163x35)
    Ellipse (579,156 25x25)
    Ellipse (660,156 25x25)
    Ellipse (616,163 10x10)
    Ellipse (638,163 10x10)
    Label (559,186 64x39), "USER SETTING"
    Label (640,186 64x24), "ADD USER"
    Image (514,146 45x45), image: ImagePool.Previous Button
        OnMouseClick: change screen: UserSetting_Page
    Group (1155,740 61x86)
        toggle bUM_CreatePB
        Button (8,0 45x45)
        Label (0,44 61x42), "CREATE USER"
        Image (14,9 32x27), image: ImagePool.Add User
    Group (1242,740 60x80)
        toggle bUM_ReturnPB
        Button (8,0 45x45)
        Label (0,36 60x44), "CANCEL"
        Image (15,5 30x35), image: ImagePool.Cancel
    Rectangle (155,558 515x30), "%s", text variable: sUM_NewUserFirstName
        OnMouseDown: write the text variable via Default
    Rectangle (156,659 515x30), "%s", text variable: sUM_NewUserLastName
        OnMouseDown: write the text variable via Default
    Rectangle (154,460 515x30), "%s", text variable: sUM_NewUserLoginName
        OnMouseDown: write the text variable via Default
    Textfield (158,374 768x30), "%s", text variable: sMessage
    Frame (0,84 1918x221), invisible if: HMI_Ctrl.CloseMenuButton
        shows Popup_MenuPage()
END_VISUALIZATION

// ---- VISUs/USER_SETTING/Edit_User.TcVIS
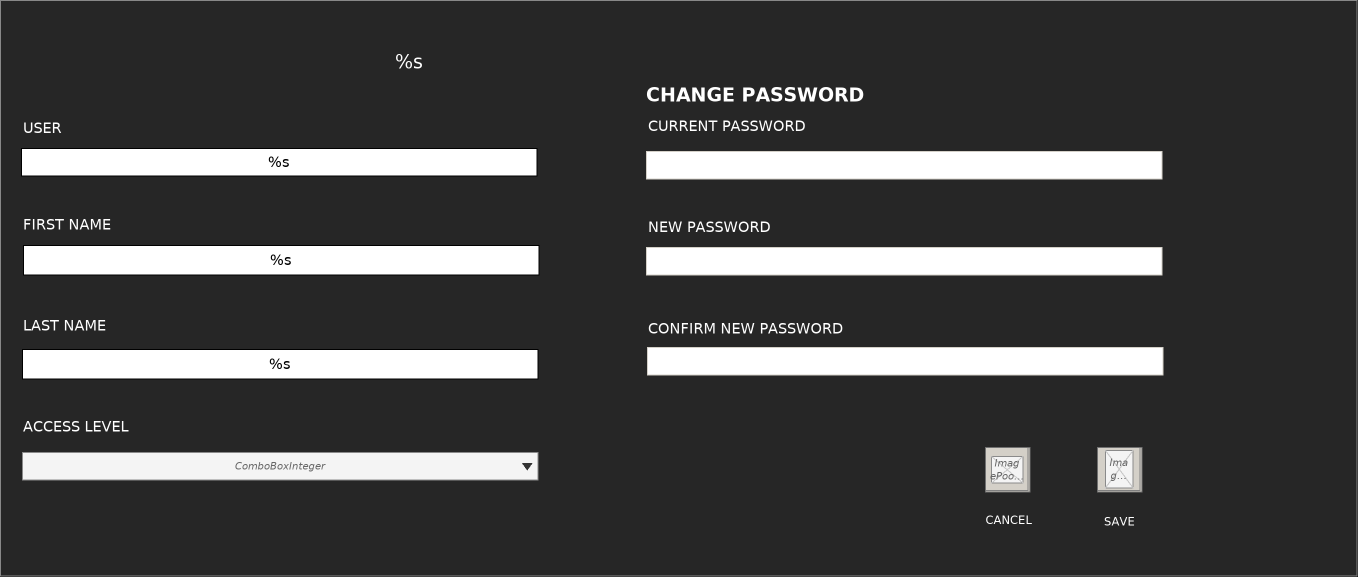
VISUALIZATION Edit_User  // 1358x577
    Rectangle (0,0 1358x577)
    Label (20,400 216x53), "ACCESS LEVEL"
    Label (20,299 216x53), "LAST NAME"
    Label (20,97 123x62), "USER"
    Label (20,198 216x53), "FIRST NAME"
    Label (643,76 417x38), "CHANGE PASSWORD"
    Label (645,196 195x62), "NEW PASSWORD"
    Label (645,302 230x53), "CONFIRM NEW PASSWORD"
    Textfield (647,347 516x28), text variable: sUM_ConfirmPassword
        OnMouseDown: write the text variable via Default, password
    Textfield (646,247 516x28), text variable: sUM_NewPassword
        OnMouseDown: write the text variable via Default, password
    Group (1077,447 85x99)
        toggle bUM_ConfirmPB
        OnMouseDown: toggle bUserNameEditPageOn
        Button (20,0 45x45)
        Label (0,50 85x49), "SAVE"
        Image (28,3 28x38), image: ImagePool.Save Button
    Group (954,447 110x102)
        toggle bUM_ReturnPB
        OnMouseDown: toggle bUserNameEditPageOn
        Button (31,0 45x45)
        Label (0,44 110x58), "CANCEL"
        Image (37,9 32x27), image: ImagePool.Delete User
    Label (645,95 195x62), "CURRENT PASSWORD"
    Textfield (646,151 516x28), text variable: sUM_CurrentPassword
        OnMouseDown: write the text variable via Default, password
    Rectangle (21,148 516x28), "%s", text variable: sUM_NewUserFirstName
        OnMouseDown: write the text variable via Default
    Rectangle (23,245 516x30), "%s", text variable: sUM_NewUserFirstName
        OnMouseDown: write the text variable via Default
    Rectangle (22,349 516x30), "%s", text variable: sUM_NewUserLastName
        OnMouseDown: write the text variable via Default
    Textfield (25,47 768x30), "%s", text variable: sMessage
    ComboBoxInteger (22,452 516x28), variable: sUM_NewUserGroupId, text list: 'TextList_AccessLevel'
END_VISUALIZATION

// ---- VISUs/USER_SETTING/UserSetting_Page.TcVIS
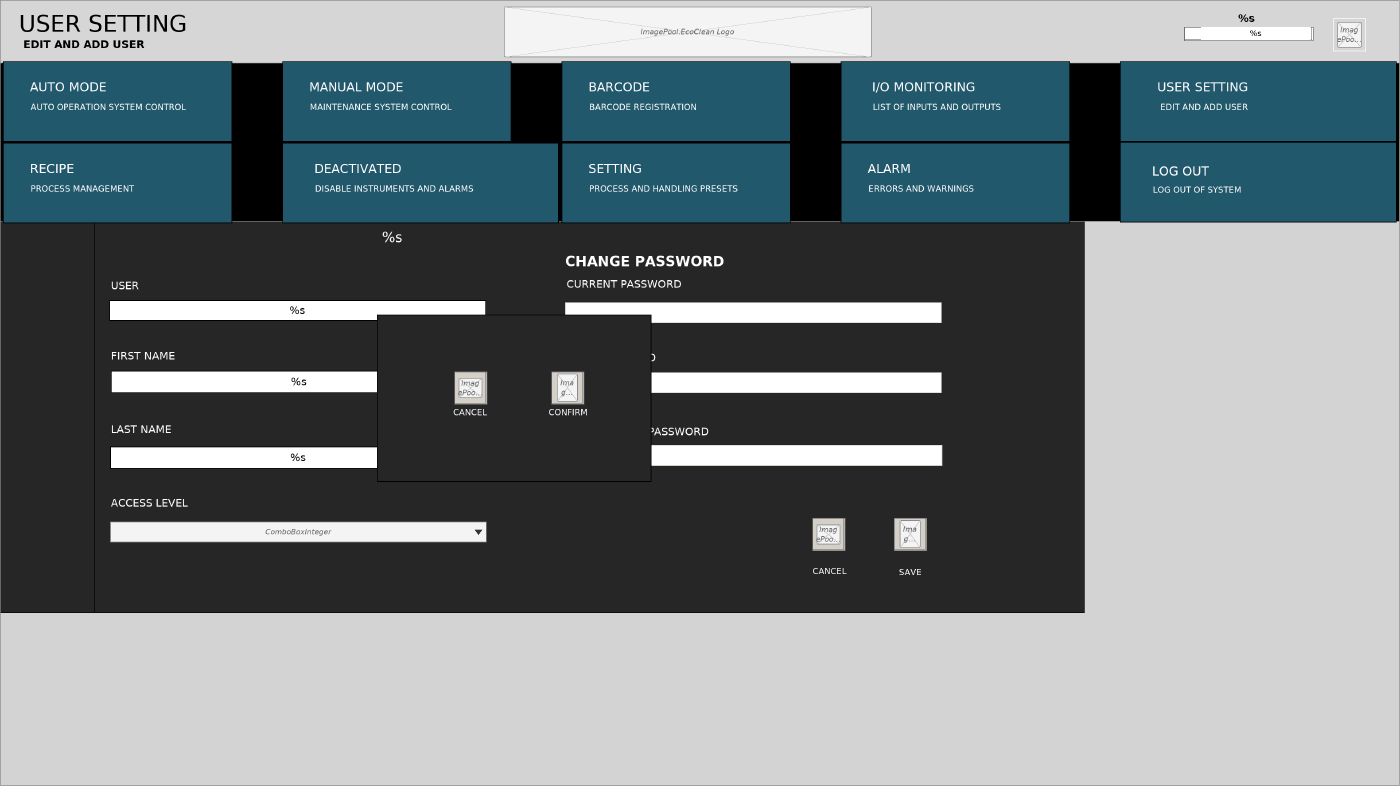
VISUALIZATION UserSetting_Page  // 1920x1079
    Rectangle (0,98 1920x981)
    Rectangle (0,63 1920x26)
        p3528305787: HMI_Ctrl.ANIMATION3
    Rectangle (0,0 1919x85)
    Label (23,6 310x53), "USER SETTING"
    Label (29,49 320x24), "EDIT AND ADD USER"
    Group (1828,25 45x45)
        OnMouseClick: toggle HMI_Ctrl.MenuButton
        RoundedRectangle (0,0 45x45), colour toggle: HMI_Ctrl.MenuButton
        Image (6,5 33x35), image: ImagePool.Menu Button
    Image (691,9 504x69), image: ImagePool.EcoClean Logo
    Group (1621,14 180x42)
        Rectangle (0,0 177x22), "%s", text variable: DSLocalSystemTimeML.sCurrentDT24Hr_General
        Button (3,23 177x19), image: VisuSymbols.Symbols.AddUser
        Rectangle (26,23 150x18), "%s", text variable: fbHmiTF1800_UserlevelManagement.dsHmiUserStatus_Active.sLoginName
    Rectangle (0,264 1358x577)
    Label (153,284 221x53), "USER SETTING"
    Label (156,321 609x38), "CHANGE USER DETAILS AND INFORMATION"
    Label (154,712 216x53), "ACCESS LEVEL"
    Label (154,611 216x53), "LAST NAME"
    Label (154,409 123x62), "USER"
    Label (154,510 216x53), "FIRST NAME"
    RoundedRectangle (550,151 162x35)
    Ellipse (579,156 25x25)
    Ellipse (660,156 25x25)
    Ellipse (616,163 10x10)
    Ellipse (638,163 10x10)
    Label (559,186 64x39), "USER SETTING"
    Label (640,186 64x24), "ADD USER"
    Image (717,146 45x45), image: ImagePool.Next Button
        OnMouseClick: change screen: AddNewUser_Page
    Group (699,739 60x88)
        toggle bUM_EditPB
        OnMouseDown: toggle bUserNameEditPageOn
        OnMouseDown: toggle bUM_EditPB
        Button (8,0 45x45)
        Label (0,44 60x44), "EDIT"
        Image (14,9 32x27), image: ImagePool.Delete User
    Group (155,460 516x28)
        toggle bUserNameLoginPageOn
        Rectangle (0,0 516x28), "%s", text variable: fbHmiTF1800_UserlevelManagement.dsHmiUserReg.ARsLoginName[iUM_SelectedLoginNameId]
        Group (481,0 35x28)
            Rectangle (0,0 40x34)
            Image (4,2 32x32), image: VisuSymbols.Symbols.TriangleDown
    Rectangle (157,557 516x30), "%s", text variable: fbHmiTF1800_UserlevelManagement.dsHmiUserReg.ARsFirstName[iUM_SelectedLoginNameId]
        OnMouseDown: write the text variable via Default
    Rectangle (156,661 516x30), "%s", text variable: fbHmiTF1800_UserlevelManagement.dsHmiUserReg.ARsLastName[iUM_SelectedLoginNameId]
        OnMouseDown: write the text variable via Default
    Textfield (159,359 768x30), "%s", text variable: sMessage
    Table (157,488 512x130), invisible if: NOT bUserNameLoginPageOn, data array: fbHmiTF1800_UserlevelManagement.dsHmiUserReg.ARsLoginName
        p1137915858: iUM_SelectedLoginNameId
        p3854506369: fbHmiTF1800_UserlevelManagement.dsHmiUserReg.ARsLoginName[INDEX]
        p2232123230: Login Name
        Columns.Column.[0].Template: toggle bUserNameLoginPageOn
    Rectangle (156,757 513x30), "%s", text variable: fbHmiTF1800_UserlevelManagement.dsHmiUserReg.ARwsUserGroupName[iUM_SelectedLoginNameId]
    Group (765,740 60x88)
        toggle bUM_DeletePB
        Button (8,0 45x45)
        Label (0,44 60x44), "DELETE"
        Image (14,9 32x27), image: ImagePool.Delete User
    Frame (129,264 1376x450), invisible if: NOT bUserNameEditPageOn
        shows Edit_User()
    Group (517,432 376x229), invisible if: NOT bPageConfirmPageOn
        Rectangle (0,0 376x229)
        Group (230,78 65x68)
            toggle bUM_ConfirmPB
            Button (9,0 45x45)
            Label (0,44 65x24), "CONFIRM"
            Image (17,3 28x38), image: ImagePool.Save Button
        Group (98,78 60x78)
            toggle bUM_ReturnPB
            OnMouseDown: toggle bPageConfirmPageOn
            Button (8,0 45x45)
            Label (0,34 60x44), "CANCEL"
            Image (14,9 32x27), image: ImagePool.Delete User
    Frame (0,84 1918x221), invisible if: HMI_Ctrl.CloseMenuButton
        shows Popup_MenuPage()
END_VISUALIZATION

// ---- VISUs/Vertical_Arm_Traveling_Zone.TcVIS
VISUALIZATION Vertical_Arm_Traveling_Zone  // 2x2
END_VISUALIZATION

// ---- VISUs/Visualization.TcVIS
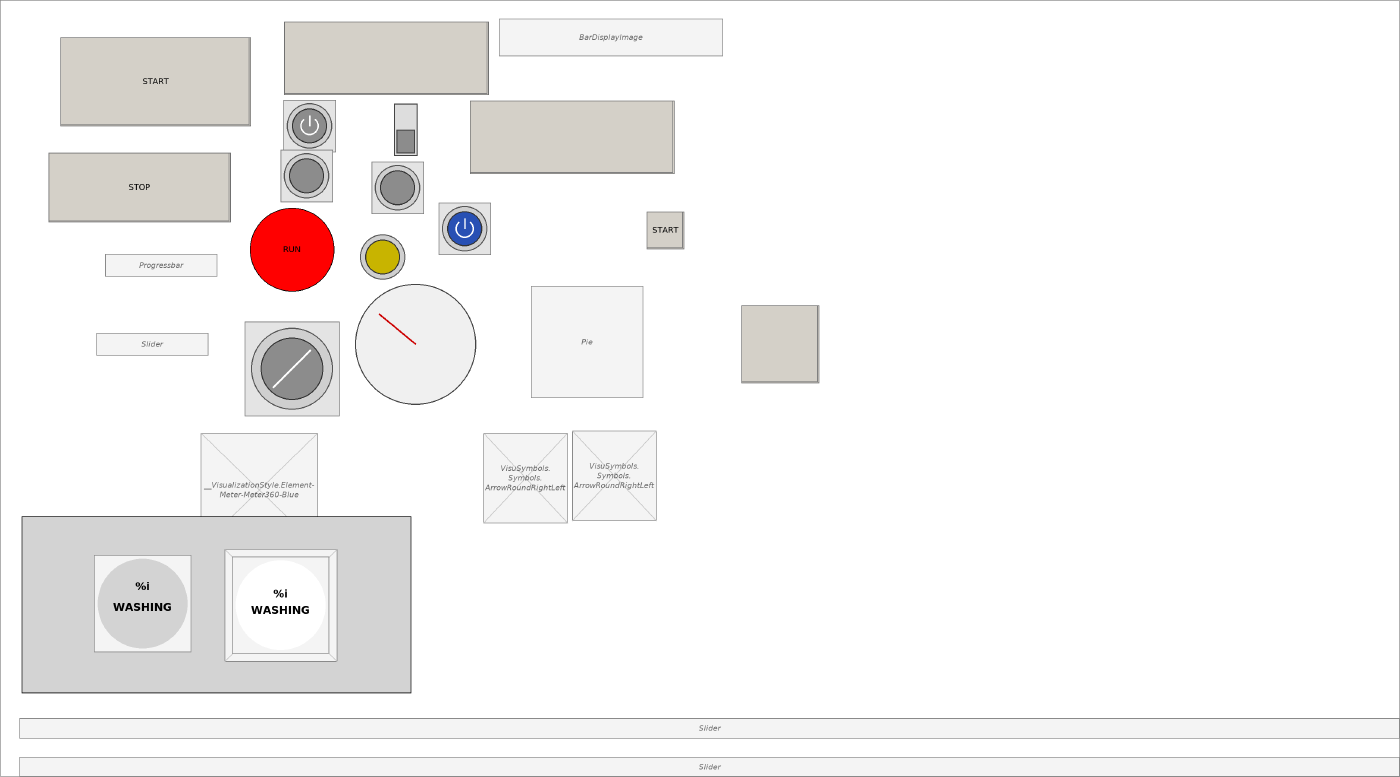
VISUALIZATION Visualization  // 1877x1043
    Button (81,50 255x119), "START"
        tap StartStop.Start
    Button (65,205 244x93), "STOP"
        tap StartStop.Stop
    DipSwitch (509,139 70x70), variable: StartStop.Start, behaviour: TOGGLE, style: Switch-DipSwitch-Gray
    Lamp1 (478,310 70x70), variable: StartStop.Run, style: Lamp-Lamp1-Yellow
    PowerSwitch (380,134 70x70), variable: StartStop.Start, behaviour: TOGGLE, style: Switch-PowerSwitch-Gray
    PushSwitch (376,201 70x70), variable: StartStop.Start, behaviour: TOGGLE, style: Switch-PushSwitch-Gray
    PushSwitchLed (498,217 70x70), variable: StartStop.Start, behaviour: TOGGLE, style: Switch-PushSwitchLed-Gray
    RockerSwitch (476,46 70x70), variable: StartStop.Start, behaviour: TOGGLE, style: Switch-RockerSwitch-Gray
    RotarySwitch (571,43 70x70), variable: StartStop.Start, behaviour: TOGGLE, style: Switch-RotarySwitch-Gray
    BarDisplayImage (669,25 300x50), value: StartStop.Value, style: BarDisplayImage-Gray, scale format: %.1f, scale 0..100
    Meter360 (476,379 162x166), value: StartStop.Value, style: Meter-Meter360-Gray, scale format: %.1f, scale 0..100
    Potentiometer360 (328,427 127x136), variable: StartStop.Value, style: Potentiometer-Potentiometer360-Gray, scale format: %.1f, scale 0..100
        p2431819421: Outside
    Progressbar (141,341 150x30), variable: StartStop.Value
    Slider (129,447 150x30), variable: StartStop.Value, scale 0..100
    Pie (712,384 150x150)
        p426801730: StartStop.Value
    Image (269,581 157x153)
        p573394764: StartStop.Value
    Ellipse (335,279 113x112), "RUN", colour toggle: StartStop.Run
    PowerSwitch (588,272 70x70), variable: StartStop.Start, behaviour: TOGGLE, style: Switch-PowerSwitch-Blue
    Image (648,581 113x121), image: VisuSymbols.Symbols.ArrowRoundRightLeft
        p2277200375: StartStop.Value
    Image (767,578 113x121), image: VisuSymbols.Symbols.ArrowRoundRightLeft
        p2858320360: StartStop.Value
    Button (630,135 274x98)
        OnMouseClick: toggle StartStop.Stop
    Button (381,29 274x98)
        OnMouseClick: change screen: Login_Page
    Button (867,284 50x50), "START", image: VisuSymbols.Symbols.TriangleDown
        tap StartStop.Start
    Rectangle (29,693 522x237)
    Pie (126,745 130x130)
        p426801730: StartStop.Value
        p2124672552: StartStop.FAIZValue2
    Ellipse (131,750 120x120), colour toggle: StartStop.Start
        toggle StartStop.Start
    Label (171,782 40x24)
    Label (150,803 82x24), "WASHING"
    Image (301,737 151x151)
        p573394764: StartStop.Value
    Pie (311,747 130x130)
        p426801730: StartStop.Value
        p2124672552: StartStop.FAIZValue2
    Ellipse (316,752 120x120), colour toggle: StartStop.Start
        toggle StartStop.Start
    Rectangle (342,782 69x30), "%i", text variable: StartStop.Value
    Rectangle (157,772 69x30), "%i", text variable: StartStop.Value
    Label (335,807 82x24), "WASHING"
    Slider (26,964 1851x27), variable: StartStop.Value, scale 0..360
    Slider (26,1016 1851x27), variable: StartStop.FAIZValue2, scale 0..360
    Button (994,410 104x104)
END_VISUALIZATION
